# EPICS substitutions: iocBoot/iocalvsvr/alive.substitutions
file "$(TOP)/db/aliverec.db" { pattern
{  BL,    DEV,              R, HMAG, DEADTIME}
{PINK, ALVSRV,    aliveclient,    0,       10}
}
